FUNCTION_BLOCK DualHysteresis_AR_AX (* 2-way conversion of Analog to Digital with Hysteresis *)
  (* Standard: 61499-2; Description: Copyright (c) 2023 HR Agrartechnik GmbH This program and the accompanying materials are made available under the terms of the Eclipse Public License 2.0 which is available at https://www.eclipse.org/legal/epl-2.0/ SPDX-License-Identifier: EPL-2.0 *)
  (* Version 3.0, 2025-04-14, Patrick Aigner, changed package *)
  (* Version 1.0, 2023-06-06, Franz Höpfinger, HR Agrartechnik GmbH *)
  PACKAGE logiBUS::signalprocessing;
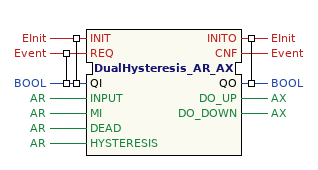
  EVENT_INPUT
    INIT : EInit WITH QI; (* Initialization Request *)
    REQ WITH QI; (* Normal Execution Request *)
  END_EVENT
  EVENT_OUTPUT
    INITO : EInit WITH QO; (* Initialization Confirm *)
    CNF; (* Execution Confirmation *)
  END_EVENT
  VAR_INPUT
    QI : BOOL; (* Input event qualifier *)
  END_VAR
  VAR_OUTPUT
    QO : BOOL;
  END_VAR
  SOCKETS
    INPUT : adapter::types::unidirectional::AR; (* Input value *)
    MI : adapter::types::unidirectional::AR; (* MID Setting can e.g. be 0.5 meaning 50% *)
    DEAD : adapter::types::unidirectional::AR; (* Deadband around MID can be e.g. 0.1 meaning 10% *)
    HYSTERESIS : adapter::types::unidirectional::AR; (* Hysteresis can be 0.1 meaning 10% *)
  END_SOCKETS
  PLUGS
    DO_UP : adapter::types::unidirectional::AX; (* UP *)
    DO_DOWN : adapter::types::unidirectional::AX; (* DOWN *)
  END_PLUGS
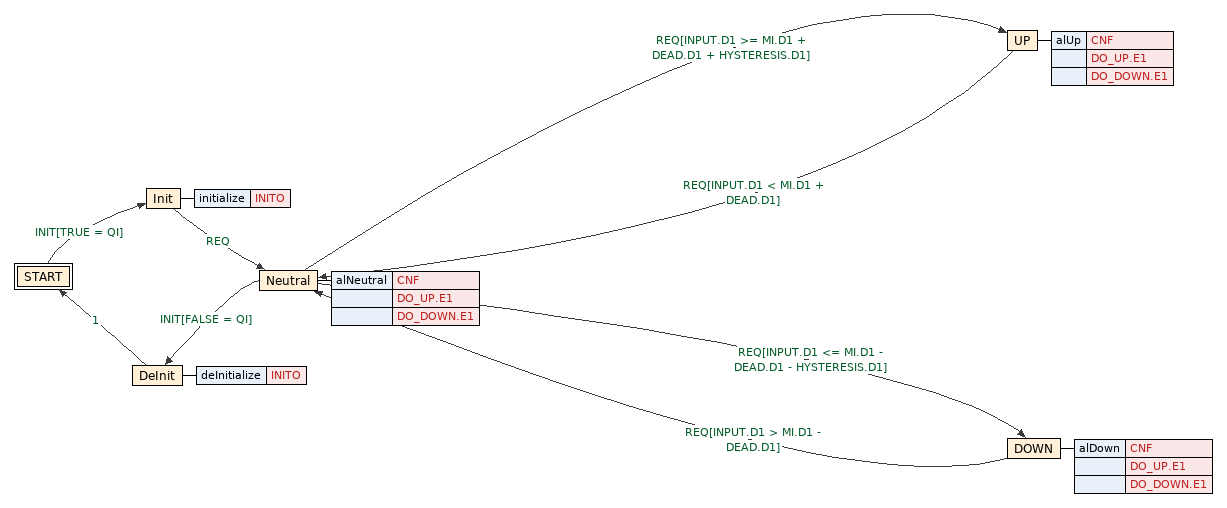
  EC_STATES
    START; (* Initial State *)
    Init : initialize -> INITO; (* Initialization *)
    UP : alUp -> CNF, -> DO_UP.E1, -> DO_DOWN.E1; (* Normal execution *)
    Neutral : alNeutral -> CNF, -> DO_UP.E1, -> DO_DOWN.E1;
    DeInit : deInitialize -> INITO;
    DOWN : alDown -> CNF, -> DO_UP.E1, -> DO_DOWN.E1;
  END_STATES
  EC_TRANSITIONS
    START TO Init := INIT[TRUE = QI];
    Init TO Neutral := REQ;
    Neutral TO DeInit := INIT[FALSE = QI];
    Neutral TO UP := REQ[INPUT.D1 >= MI.D1 + DEAD.D1 + HYSTERESIS.D1];
    DeInit TO START := 1;
    Neutral TO DOWN := REQ[INPUT.D1 <= MI.D1 - DEAD.D1 - HYSTERESIS.D1];
    DOWN TO Neutral := REQ[INPUT.D1 > MI.D1 - DEAD.D1];
    UP TO Neutral := REQ[INPUT.D1 < MI.D1 + DEAD.D1];
  END_TRANSITIONS
  ALGORITHM initialize IN ST:
QO := QI;
(* in any case go safe State *)
DO_UP.D1 := BOOL#FALSE;
DO_DOWN.D1 := BOOL#FALSE;
  END_ALGORITHM
  ALGORITHM deInitialize IN ST:
QO := BOOL#FALSE;
(* in any case go safe State *)
DO_UP.D1 := BOOL#FALSE;
DO_DOWN.D1 := BOOL#FALSE;
  END_ALGORITHM
  ALGORITHM alNeutral IN ST:
QO := QI;
(* in any case go safe State *)
DO_UP.D1 := BOOL#FALSE;
DO_DOWN.D1 := BOOL#FALSE;
  END_ALGORITHM
  ALGORITHM alUp IN ST:
QO := QI;
IF TRUE = QI THEN
	(* only perform normal operation of QI is true *)
	DO_UP.D1 := BOOL#TRUE;
	DO_DOWN.D1 := BOOL#FALSE;
END_IF;
  END_ALGORITHM
  ALGORITHM alDown IN ST:
QO := QI;
IF TRUE = QI THEN
	(* only perform normal operation of QI is true *)
	DO_UP.D1 := BOOL#FALSE;
	DO_DOWN.D1 := BOOL#TRUE;
END_IF;
  END_ALGORITHM
END_FUNCTION_BLOCK
